# EPICS autosave request: trunk/mcaApp/Db/Struck_settings.req
$(P)PresetReal
$(P)Dwell
$(P)Prescale
$(P)ChannelAdvance
$(P)StatusAll.SCAN
$(P)ReadAll.SCAN
$(P)NuseAll
$(P)EnableClientWait
